TYPE T_Ctrl_SIf_AGS_Cfg :
STRUCT
END_STRUCT
END_TYPE

(* stored: Version 1.1.0.1, ProductVersion 3.1.0.26
   DUT T_Ctrl_SIf_AGS_Cfg: Id {842b0f51-3f0e-4d69-ab76-2b47821e5188} *)
